% RSLogix 500 project PLC1_L2-2B.RSS, saved by version 12.00.00.00 %
PROJECT "UNTITLED"    % processor: Bul.1763 MicroLogix 1100 Series B %

PROGRAM FILES
  LAD 2   2 rungs

DATA FILES
  O0 OUTPUT  5 elements
  I1 INPUT  6 elements
  S2 STATUS  66 elements
  B3 BINARY  1 elements
  T4 TIMER  1 elements
  C5 COUNTER  1 elements
  R6 CONTROL  1 elements
  N7 INTEGER  1 elements
  F8 FLOAT  1 elements

LADDER 2
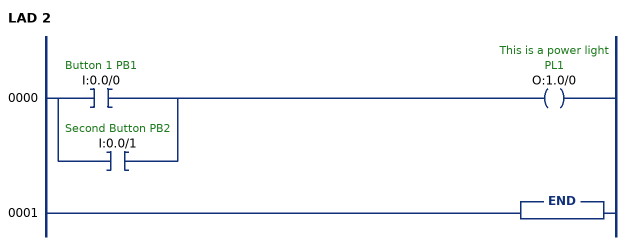
% Rung: 0 %
SOR BST XIC I:0.0/0 NXB XIC I:0.0/1 BND OTE O:1.0/0 EOR
%   I:0.0/0  PB1  "Button 1" %
%   I:0.0/1  PB2  "Second Button" %
%   O:1.0/0  PL1  "This is a power light" %
% Rung: 1 %
SOR END EOR

REVISION NOTES
  0: last change
  1: Lab2-2b
